// TIA Portal V18 export
DATA_BLOCK "SS1_A3_8xAI_AI_Vars"   // DB11031
{ S7_Optimized_Access := 'FALSE' }
VERSION : 0.1
// stored: AutoNumber false, DBAccessibleFromOPCUA true, IsOnlyStoredInLoadMemory false, IsWriteProtectedInAS false
   VAR
      AI1 { S7_SetPoint := 'True'} : "UDT_AIadv";
      AI2 { S7_SetPoint := 'True'} : "UDT_AIadv";
      AI3 { S7_SetPoint := 'True'} : "UDT_AIadv";
      AI4 { S7_SetPoint := 'True'} : "UDT_AIadv";
      AI5 { S7_SetPoint := 'True'} : "UDT_AIadv";
      AI6 { S7_SetPoint := 'True'} : "UDT_AIadv";
      AI7 { S7_SetPoint := 'True'} : "UDT_AIadv";
      AI8 { S7_SetPoint := 'True'} : "UDT_AIadv";
   END_VAR
BEGIN
   AI1.rValue := 0.3255208;
   AI1.rMin := 0.0;
   AI1.rMax := 1000.0;
   AI1.rCalibration := 0.0;
   AI1.iFuncSystemID := 16#00;
   AI1.iFuncVar := 16#00;
   AI1.rFilterSet := 0.0;
   AI2.rValue := 1.808449;
   AI2.rMin := 0.0;
   AI2.rMax := 1000.0;
   AI2.rCalibration := 0.0;
   AI2.iFuncSystemID := 16#00;
   AI2.iFuncVar := 16#00;
   AI2.rFilterSet := 0.0;
   AI3.rValue := 3.616898E-05;
   AI3.rMin := 0.0;
   AI3.rMax := 0.0;
   AI3.rCalibration := 0.0;
   AI3.iFuncSystemID := 16#00;
   AI3.iFuncVar := 16#00;
   AI3.rFilterSet := 0.0;
   AI4.rValue := 0.0003255208;
   AI4.rMin := 0.0;
   AI4.rMax := 0.0;
   AI4.rCalibration := 0.0;
   AI4.iFuncSystemID := 16#00;
   AI4.iFuncVar := 16#00;
   AI4.rFilterSet := 0.0;
   AI5.rValue := 6.04022;
   AI5.rMin := 0.0;
   AI5.rMax := 1000.0;
   AI5.rCalibration := 0.0;
   AI5.iFuncSystemID := 16#01;
   AI5.iFuncVar := 16#0A;
   AI5.rFilterSet := 0.0;
   AI6.rValue := 17.15549;
   AI6.rMin := 0.0;
   AI6.rMax := 15.0;
   AI6.rCalibration := 0.0;
   AI6.iFuncSystemID := 16#01;
   AI6.iFuncVar := 16#07;
   AI6.rFilterSet := 0.0;
   AI7.rValue := 29.49942;
   AI7.rMin := 0.0;
   AI7.rMax := 100.0;
   AI7.rCalibration := 0.0;
   AI7.iFuncSystemID := 16#00;
   AI7.iFuncVar := 16#00;
   AI7.rFilterSet := 0.0;
   AI8.rValue := 0.07957176;
   AI8.rMin := 0.0;
   AI8.rMax := 100.0;
   AI8.rCalibration := 0.0;
   AI8.iFuncSystemID := 16#00;
   AI8.iFuncVar := 16#00;
   AI8.rFilterSet := 0.0;
END_DATA_BLOCK
